(* CODESYS project BagFeedMotorTest.xml

Project tree, tasks and I/O mapping:
  program BagFeedMotorTest [LD]
*)

// BagFeedMotorTest
PROGRAM BagFeedMotorTest
VAR_INPUT
END_VAR
VAR_OUTPUT
END_VAR
VAR
END_VAR

// NETWORK 1

END_PROGRAM
